// Mitsubishi GX Works2 project: Class6_Moter&Cylinder&Conveyor   PLC: Q03UD

PROGRAM Cylinder
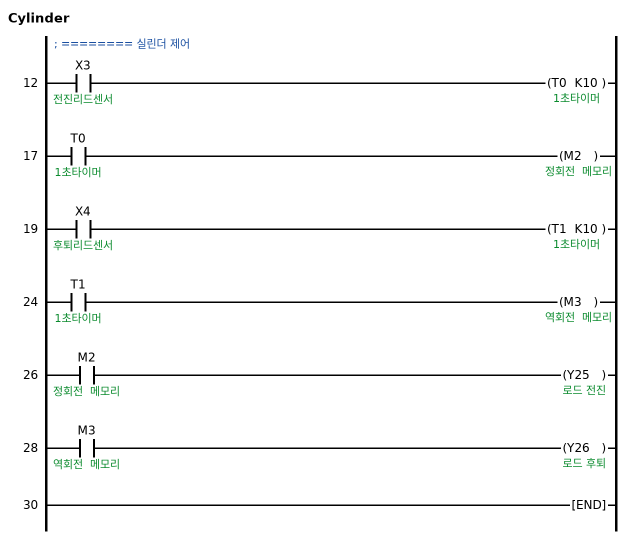
; ======== 실린더 제어
12    LD      X3  ; 전진리드센서
      OUT     T0 K10  ; 1초타이머
17    LD      T0  ; 1초타이머
      OUT     M2  ; 정회전  메모리
19    LD      X4  ; 후퇴리드센서
      OUT     T1 K10  ; 1초타이머
24    LD      T1  ; 1초타이머
      OUT     M3  ; 역회전  메모리
26    LD      M2  ; 정회전  메모리
      OUT     Y25  ; 로드 전진
28    LD      M3  ; 역회전  메모리
      OUT     Y26  ; 로드 후퇴
30    END
END_PROGRAM

PROGRAM Conveyor
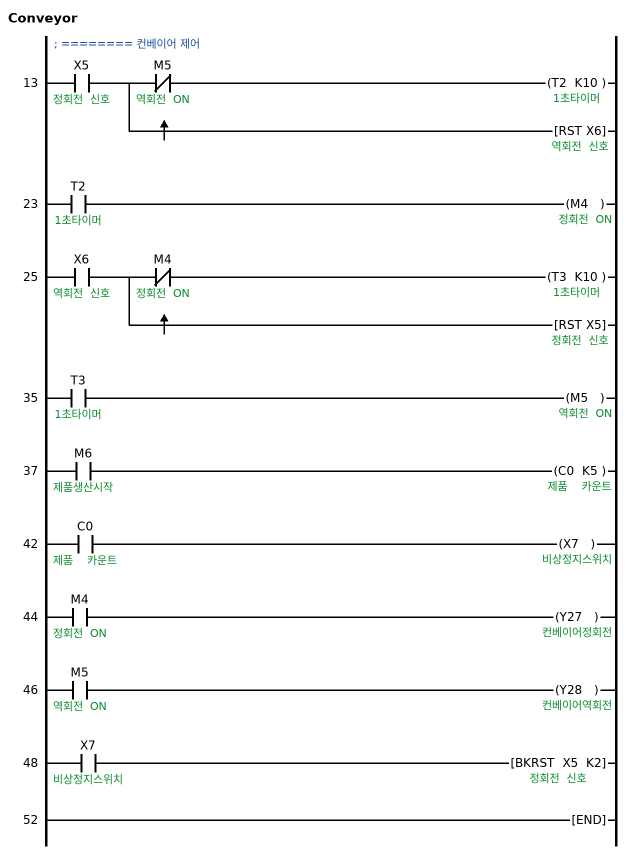
; ======== 컨베이어 제어
13    LD      X5  ; 정회전  신호
      MPS
      ANI     M5  ; 역회전  ON
      OUT     T2 K10  ; 1초타이머
      MPP
      MEP
      RST     X6  ; 역회전  신호
23    LD      T2  ; 1초타이머
      OUT     M4  ; 정회전  ON
25    LD      X6  ; 역회전  신호
      MPS
      ANI     M4  ; 정회전  ON
      OUT     T3 K10  ; 1초타이머
      MPP
      MEP
      RST     X5  ; 정회전  신호
35    LD      T3  ; 1초타이머
      OUT     M5  ; 역회전  ON
37    LD      M6  ; 제품생산시작
      OUT     C0 K5  ; 제품    카운트
42    LD      C0  ; 제품    카운트
      OUT     X7  ; 비상정지스위치
44    LD      M4  ; 정회전  ON
      OUT     Y27  ; 컨베이어정회전
46    LD      M5  ; 역회전  ON
      OUT     Y28  ; 컨베이어역회전
48    LD      X7  ; 비상정지스위치
      BKRST   X5 K2
52    END
END_PROGRAM

PROGRAM ACMotor
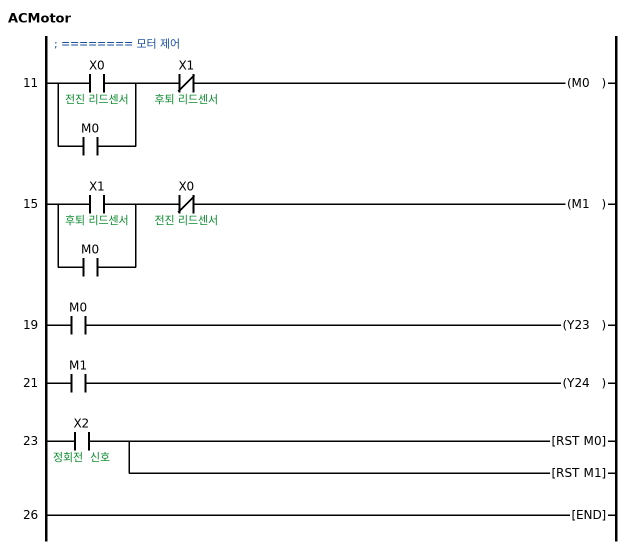
; ======== 모터 제어
11    LD      X0  ; 전진 리드센서
      OR      M0
      ANI     X1  ; 후퇴 리드센서
      OUT     M0
15    LD      X1  ; 후퇴 리드센서
      OR      M0
      ANI     X0  ; 전진 리드센서
      OUT     M1
19    LD      M0
      OUT     Y23
21    LD      M1
      OUT     Y24
23    LD      X2  ; 정회전  신호
      RST     M0
      RST     M1
26    END
END_PROGRAM

// device comments not shown above
M7  ; 정회전  중지
